RESOURCE_TYPE topFLAT
  (* Standard: 61499-2 *)
  (* Version 0.1, 2017-00-09, Hammond, HAMMONDSDESKTOP *)
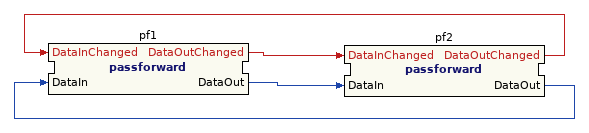
  FBS
    pf1 : passforward;
    pf2 : passforward;
  END_FBS
  EVENT_CONNECTIONS
    pf1.DataOutChanged TO pf2.DataInChanged;
    pf2.DataOutChanged TO pf1.DataInChanged;
  END_CONNECTIONS
  DATA_CONNECTIONS
    pf1.DataOut TO pf2.DataIn;
    pf2.DataOut TO pf1.DataIn;
  END_CONNECTIONS
END_RESOURCE_TYPE
